// TIA Portal V19 export
TYPE "LAF_typeXXXParameters"
// stored: Access Published
   STRUCT
      cm2Axis : "LAF_typeAxisParameters";
      cm3NgStrap : "LAF_typeNgStrapParameters";
   END_STRUCT;
END_TYPE
